PROGRAM Stn1DosingPumpCtrl

VAR
END_VAR

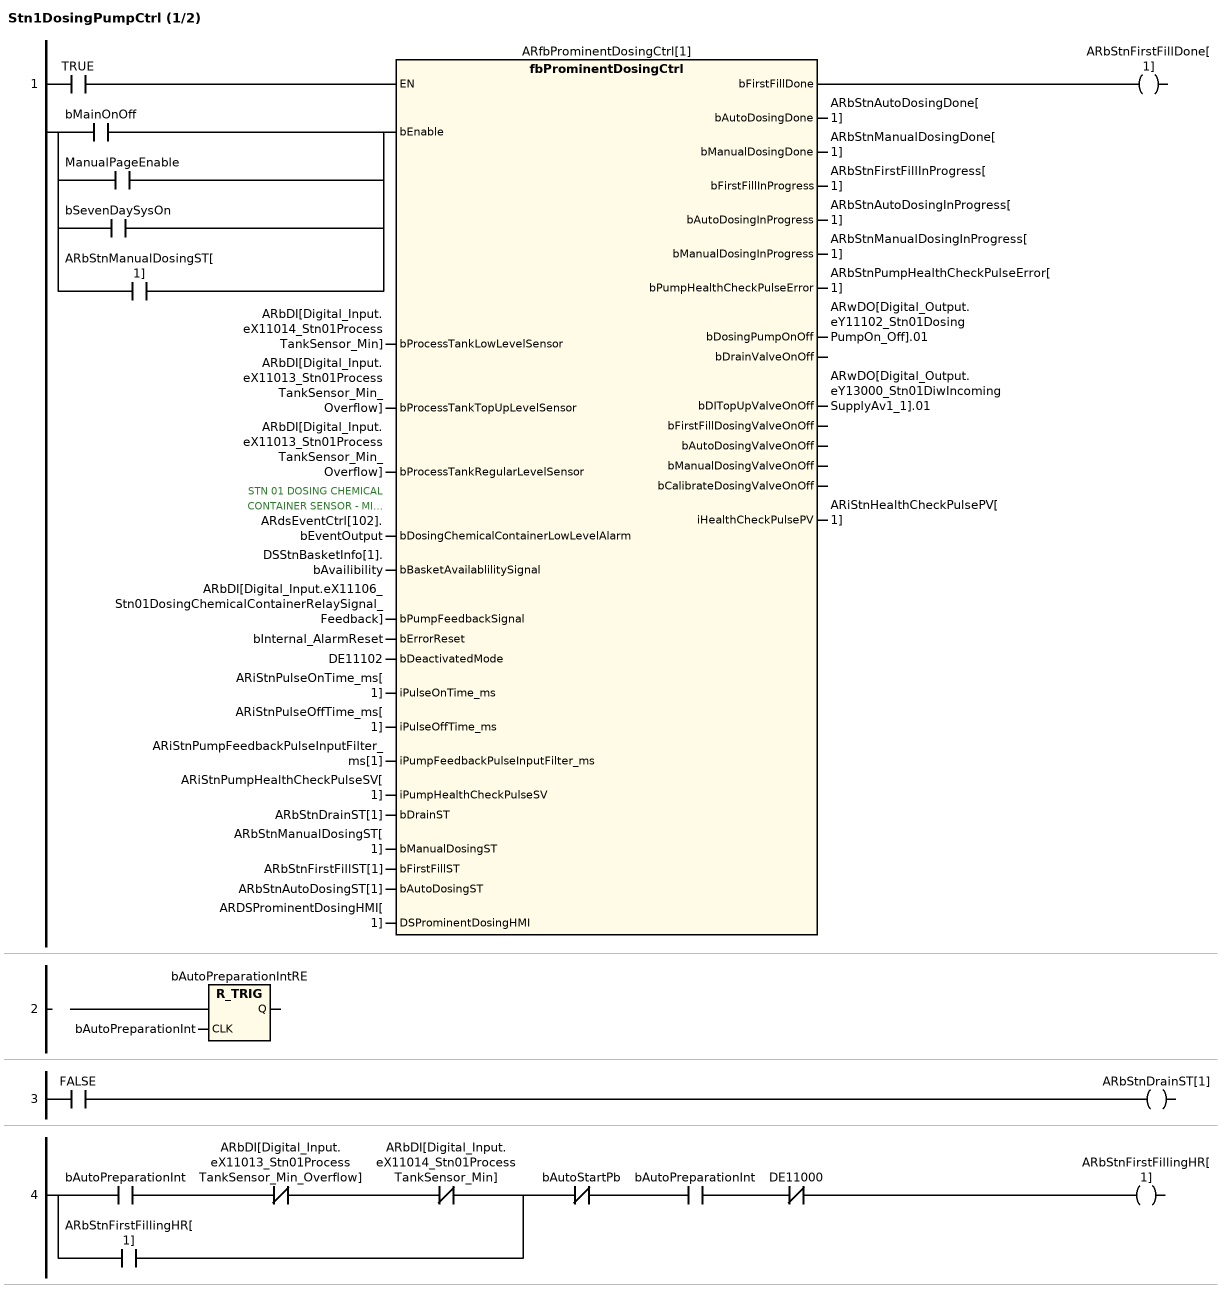
// NETWORK 1
//   ARdsEventCtrl[102].bEventOutput: STN 01 DOSING CHEMICAL CONTAINER SENSOR - MIN LEVEL
ARfbProminentDosingCtrl[1](
    bEnable := bMainOnOff OR ManualPageEnable OR bSevenDaySysOn OR ARbStnManualDosingST[1],
    bProcessTankLowLevelSensor := ARbDI[Digital_Input.eX11014_Stn01ProcessTankSensor_Min],
    bProcessTankTopUpLevelSensor := ARbDI[Digital_Input.eX11013_Stn01ProcessTankSensor_Min_Overflow],
    bProcessTankRegularLevelSensor := ARbDI[Digital_Input.eX11013_Stn01ProcessTankSensor_Min_Overflow],
    bDosingChemicalContainerLowLevelAlarm := ARdsEventCtrl[102].bEventOutput,
    bBasketAvailablilitySignal := DSStnBasketInfo[1].bAvailibility,
    bPumpFeedbackSignal := ARbDI[Digital_Input.eX11106_Stn01DosingChemicalContainerRelaySignal_Feedback],
    bErrorReset := bInternal_AlarmReset,
    bDeactivatedMode := DE11102,
    iPulseOnTime_ms := ARiStnPulseOnTime_ms[1],
    iPulseOffTime_ms := ARiStnPulseOffTime_ms[1],
    iPumpFeedbackPulseInputFilter_ms := ARiStnPumpFeedbackPulseInputFilter_ms[1],
    iPumpHealthCheckPulseSV := ARiStnPumpHealthCheckPulseSV[1],
    bDrainST := ARbStnDrainST[1],
    bManualDosingST := ARbStnManualDosingST[1],
    bFirstFillST := ARbStnFirstFillST[1],
    bAutoDosingST := ARbStnAutoDosingST[1],
    DSProminentDosingHMI := ARDSProminentDosingHMI[1],
    bAutoDosingDone => ARbStnAutoDosingDone[1],
    bManualDosingDone => ARbStnManualDosingDone[1],
    bFirstFillInProgress => ARbStnFirstFillInProgress[1],
    bAutoDosingInProgress => ARbStnAutoDosingInProgress[1],
    bManualDosingInProgress => ARbStnManualDosingInProgress[1],
    bPumpHealthCheckPulseError => ARbStnPumpHealthCheckPulseError[1],
    bDosingPumpOnOff => ARwDO[Digital_Output.eY11102_Stn01DosingPumpOn_Off].01,
    bDITopUpValveOnOff => ARwDO[Digital_Output.eY13000_Stn01DiwIncomingSupplyAv1_1].01,
    iHealthCheckPulsePV => ARiStnHealthCheckPulsePV[1]); // fbProminentDosingCtrl
ARbStnFirstFillDone[1] := ARfbProminentDosingCtrl[1].bFirstFillDone;

// NETWORK 2
bAutoPreparationIntRE(CLK := bAutoPreparationInt); // R_TRIG

// NETWORK 3
ARbStnDrainST[1] := FALSE;

// NETWORK 4
ARbStnFirstFillingHR[1] := (bAutoPreparationInt AND NOT ARbDI[Digital_Input.eX11013_Stn01ProcessTankSensor_Min_Overflow] AND NOT ARbDI[Digital_Input.eX11014_Stn01ProcessTankSensor_Min] OR ARbStnFirstFillingHR[1]) AND NOT bAutoStartPb AND bAutoPreparationInt AND NOT DE11000;

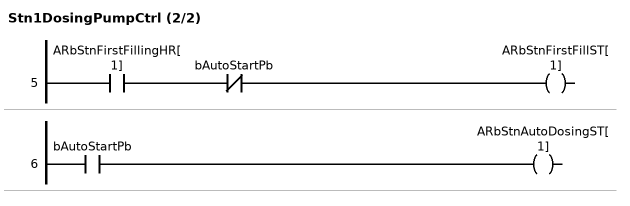
// NETWORK 5
ARbStnFirstFillST[1] := ARbStnFirstFillingHR[1] AND NOT bAutoStartPb;

// NETWORK 6
ARbStnAutoDosingST[1] := bAutoStartPb;

END_PROGRAM

(* stored: Version 1.1.0.1, ProductVersion 3.1.4024.12
   POU Stn1DosingPumpCtrl: Id {50f3d069-e859-4a65-a0bf-4057b373a3d3}, SpecialFunc None *)
